{attribute addProperty BoxType "EJ1101-0022-0016"}
{attribute addProperty Id "WcStateAT %I*WcState_28A8677510.1250InfoDataAT %I*InfoData_BC63D37F80100"}
{attribute addProperty CRC "752626490"}
{attribute addProperty SizeInBites "81"}
{attribute addProperty SizeInBytes "10.125"}
TYPE EJ1101_6969C224 :
STRUCT
	{attribute addProperty Name "WcState"}
	WcState : WcState_28A86775;
	{attribute addProperty Name "InfoData"}
	InfoData : InfoData_BC63D37F;
END_STRUCT
END_TYPE

(* stored: Version 1.2.0.0, ProductVersion 3.1.4024.9
   DUT EJ1101_6969C224: Id {c033cccb-6ee4-4f5b-8131-7d93f84e83a0} *)
